
// ===== library types =====

FUNCTION_BLOCK "MyFunctionBlock_Typed"   // FB9, FBD
TITLE = And Block
{ S7_Optimized_Access := 'TRUE' }
VERSION : 0.1
   VAR_INPUT
      Input1 : Bool;
      Input2 : Bool;
   END_VAR
   VAR_OUTPUT
      Output1 : Bool;
   END_VAR
BEGIN

REGION Network 1
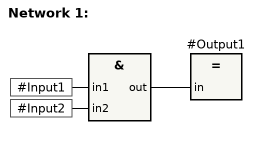
   #Output1 := #Input1 AND #Input2;
END_REGION
END_FUNCTION_BLOCK

// ===== library: MasterCopy "MyFunctionBlock" =====

FUNCTION_BLOCK "MyFunctionBlock"   // FB4, FBD
TITLE = BasicFB
{ S7_Optimized_Access := 'TRUE' }
VERSION : 0.1
   VAR_INPUT
      Input1 : Bool;
      Input2 : Bool;
   END_VAR
   VAR_OUTPUT
      Output1 : Bool;
   END_VAR
BEGIN

REGION Network 1: AndNetwork1
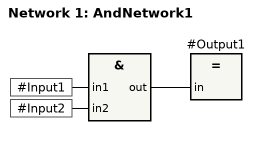
   #Output1 := #Input1 AND #Input2;
END_REGION
END_FUNCTION_BLOCK

// ===== library: MasterCopy "MyFunctionBlock_FailSafe" =====

FUNCTION_BLOCK "MyFunctionBlock_FailSafe"   // FB8, F_FBD
TITLE = FailSafe FB
{ S7_Optimized_Access := 'TRUE' }
VERSION : 0.1
   VAR_INPUT
      Input1 : Bool;
      Input2 : Bool;
   END_VAR
   VAR_OUTPUT
      Output1 : Bool;
   END_VAR
BEGIN

REGION Network 1: AndNetwork1
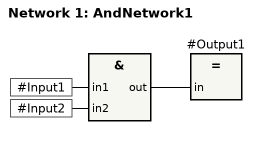
   #Output1 := #Input1 AND #Input2;
END_REGION
END_FUNCTION_BLOCK

// ===== library: MasterCopy "MyDataType" =====

TYPE "MyDataType"
   STRUCT
      myStruct : Struct
         "Int" : Int;
         "Bool" : Bool;
      END_STRUCT;
   END_STRUCT;
END_TYPE